{attribute addProperty BoxType "AMP8000-0030-0103-0103"}
{attribute addProperty Id "FSOEAT %Q*ARRAY [0..1] OF BYTE162"}
{attribute addProperty CRC "1237069497"}
{attribute addProperty SizeInBites "16"}
{attribute addProperty SizeInBytes "2"}
TYPE FSLOGIC_Outputs_49BC2EB9 :
STRUCT
	{attribute addProperty Name "FSOE"}
	FSOE AT %Q* : ARRAY [0..1] OF BYTE;
END_STRUCT
END_TYPE

(* stored: Version 1.2.0.0, ProductVersion 3.1.4024.9
   DUT FSLOGIC_Outputs_49BC2EB9: Id {d74bfb53-f457-4836-b1c7-b368ae05d6d5} *)
